{attribute 'pack_mode' := '1'}
    {attribute 'OPC.UA.DA' := '1'}
    {attribute 'OPC.UA.DA.StructuredType' := '1'}
    (*
    ST_RW_Real_Alm_HMI_IgnitionExp
    ==================================================
    Generated from Ignition UDT: RW_Real_ALM
    Total tags: 9
    Generated on: 2025-09-16 15:04:58
    *)
    TYPE ST_RW_Real_Alm_HMI_IgnitionExp :
    STRUCT
        {attribute 'OPC.UA.DA' := '1'}
        Process_Alm_Time_Hi : REAL := 0.0;
        {attribute 'OPC.UA.DA' := '1'}
        Input : REAL := 0.0;
        {attribute 'OPC.UA.DA' := '1'}
        Process_Alm_Time_LoLo : REAL := 0.0;
        {attribute 'OPC.UA.DA' := '1'}
        Process_Alm_Val_HiHi : REAL := 0.0;
        {attribute 'OPC.UA.DA' := '1'}
        Process_Alm_Val_LoLo : REAL := 0.0;

        {attribute 'OPC.UA.DA' := '1'}
        Process_Alm_Time_Lo : REAL := 0.0;
        {attribute 'OPC.UA.DA' := '1'}
        Process_Alm_Time_HiHi : REAL := 0.0;
        {attribute 'OPC.UA.DA' := '1'}
        Process_Alm_Val_Lo : REAL := 0.0;
        {attribute 'OPC.UA.DA' := '1'}
        Process_Alm_Val_Hi : REAL := 0.0;
    END_STRUCT
    END_TYPE

(* stored: Version 1.1.0.1
   DUT ST_RW_Real_Alm_HMI_IgnitionExp: Id {4b0b4c49-5b15-4900-bff7-09490ebac41a} *)
